# EPICS autosave request: 3-0/GalilSup/Db/galil_analog_out.req
$(P)$(R)_SP.VAL
$(P)$(R)_SP.DESC
$(P)$(R)_MON.DESC
